FUNCTION_BLOCK FB_RCC_TEST EXTENDS FB_TestSuite
VAR
	fbRCC : FB_RCC;
	
	stRCC_VRC_01 : ST_VRC;
	stRCC_VRC_02 : ST_VRC;
	stRCC_VRC_03 : ST_VRC;
	stRCC_VRC_04 : ST_VRC;
	stRCC_GCP_01 : ST_VG;

	
	tTimer1 : TON;
	bInitTest : BOOL := TRUE;
	xSystemOverrideMode_RCC: BOOL := FALSE;
	
	// VARS FOR TestSingleCyleExpectToTransitionThoughOneCycle
	bSeenStateZero : BOOL := FALSE;
	bSeenStateOne : BOOL := FALSE;
	bSeenStateTwo : BOOL := FALSE;
	bSeenStateThree : BOOL := FALSE;
	bSeenStateFour : BOOL := FALSE;
	bSeenStateFive : BOOL := FALSE;

END_VAR

TestSingleCyleExpectToTransitionThoughOneCycle();

METHOD TestSingleCyleExpectToTransitionThoughOneCycle : REFERENCE TO FB_Test
VAR_INPUT
END_VAR
VAR
END_VAR
TEST('TestSingleCyleExpectToTransitionThoughOneCycle');

IF bInitTest THEN
	fbRCC.start_cycle();
	bInitTest := FALSE;
	AssertEquals_INT(Expected:=-1, 
		Actual:= fbRCC.current_state, 
		Message:= 'DID NOT START AT FIRST STATE');
END_IF

tTimer1(IN:=TRUE, PT:=T#45S500ms);

// Enable RCC_VRC_03_OPEN_OK SO WE CAN MOVE ONTO NEXT STATE
(* Valve can open only when CRIX-RCC-GCP-01 reading < setpoint Torr and CRIX-RCC-VRC-01 and 04 are closed*)
IF fbRCC.current_state = 2 THEN
	stRCC_GCP_01.rPRESS := 0; 
	stRCC_GCP_01.xPRESS_OK  := TRUE;
	stRCC_VRC_01.i_xClsLS := TRUE;
	stRCC_VRC_01.q_xOPN_DO := FALSE;
	stRCC_VRC_04.i_xClsLS := TRUE;
	stRCC_VRC_04.q_xOPN_DO := FALSE;
END_IF

fbRCC(stRCC_GCP_01:=stRCC_GCP_01,
	stRCC_VRC_01:= stRCC_VRC_01,
	stRCC_VRC_02:= stRCC_VRC_02,
	stRCC_VRC_03:= stRCC_VRC_03,
	stRCC_VRC_04:= stRCC_VRC_04
);

// CHECK IF WE HAVE SEEN ALL THE STATES
IF fbRCC.current_state = 0 THEN bSeenStateZero := TRUE; END_IF
IF fbRCC.current_state = 1 THEN bSeenStateOne := TRUE; END_IF
IF fbRCC.current_state = 2 THEN bSeenStateTwo := TRUE; END_IF
IF fbRCC.current_state = 3 THEN bSeenStateThree := TRUE; END_IF
IF fbRCC.current_state = 4 THEN bSeenStateFour := TRUE; END_IF
IF fbRCC.current_state = 5 THEN bSeenStateFive :=TRUE; END_IF

		// THIS IS A TEST

				 
IF tTimer1.Q THEN
	// HAVE SE SEEN ALL STAES?
	AssertEquals_BOOL(Expected:= (bSeenStateZero AND 
									bSeenStateOne AND 
									bSeenStateTwo AND 
									bSeenStateThree AND 
									bSeenStateFour AND 
									bSeenStateFive), 
		Actual:= TRUE, 
		Message:= 'HAVE NOT VISITED ALL STATES');
	TEST_FINISHED();
	bInitTest := TRUE;
END_IF
END_METHOD

END_FUNCTION_BLOCK

(* stored: Version 1.1.0.1, ProductVersion 3.1.4024.15
   POU FB_RCC_TEST: Id {601daf38-e4c9-4c7e-b134-2d83b8bfe7a2}, SpecialFunc None
   Method TestSingleCyleExpectToTransitionThoughOneCycle: Id {3c03b652-ff1d-4d2b-b8cf-f86da69ec7c0} *)
